FUNCTION StringArrayCloseGaps : BOOL
VAR_IN_OUT
	arr : ARRAY[*] OF STRING;
END_VAR
VAR
	i : DINT;
END_VAR

END_FUNCTION

(* stored: Version 1.1.0.1, ProductVersion 3.1.4024.11
   POU StringArrayCloseGaps: Id {de20d178-933d-4650-a5be-bdde94dcce95}, SpecialFunc None *)
